FUNCTION_BLOCK oven (* ODE *)
  (* Standard: 61499-2 *)
  (* Version 0.1, 2017-00-25, hpea485, UOA *)
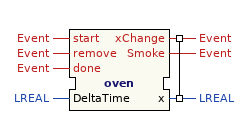
  EVENT_INPUT
    start;
    remove;
    done;
  END_EVENT
  EVENT_OUTPUT
    xChange WITH x;
    Smoke;
  END_EVENT
  VAR_INPUT
    DeltaTime : LREAL := 0.01;
  END_VAR
  VAR_OUTPUT
    x : LREAL;
  END_VAR
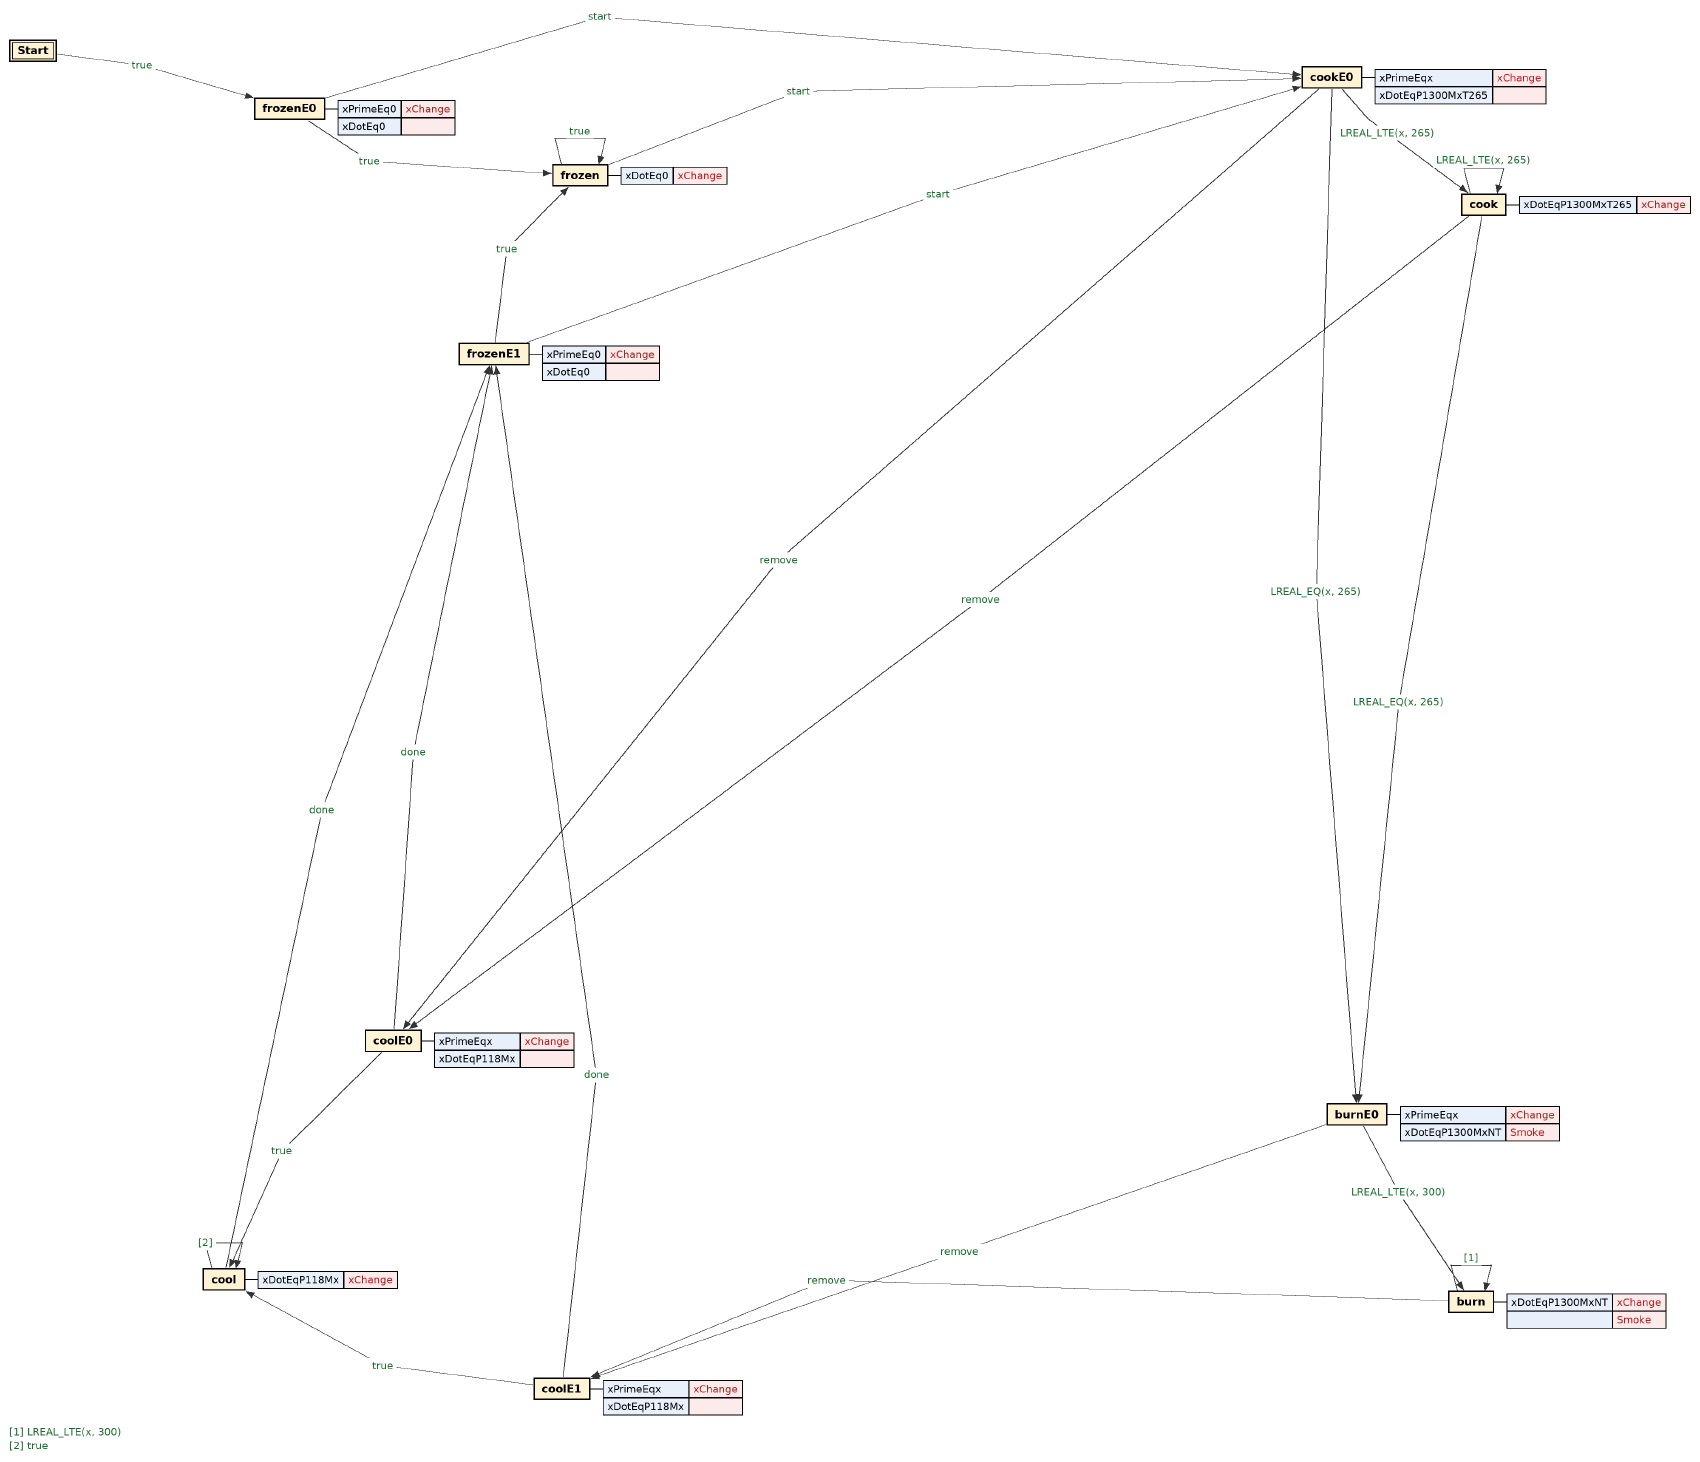
  EC_STATES
    Start;
    frozenE0 : xPrimeEq0 -> xChange, xDotEq0;
    frozen : xDotEq0 -> xChange;
    cookE0 : xPrimeEqx -> xChange, xDotEqP1300MxT265;
    cook : xDotEqP1300MxT265 -> xChange;
    burnE0 : xPrimeEqx -> xChange, xDotEqP1300MxNT -> Smoke;
    burn : xDotEqP1300MxNT -> xChange, -> Smoke;
    coolE0 : xPrimeEqx -> xChange, xDotEqP118Mx;
    coolE1 : xPrimeEqx -> xChange, xDotEqP118Mx;
    cool : xDotEqP118Mx -> xChange;
    frozenE1 : xPrimeEq0 -> xChange, xDotEq0;
  END_STATES
  EC_TRANSITIONS
    Start TO frozenE0 := true;
    frozenE0 TO cookE0 := start;
    frozenE0 TO frozen := true;
    frozen TO cookE0 := start;
    frozen TO frozen := true;
    cookE0 TO coolE0 := remove;
    cookE0 TO burnE0 := LREAL_EQ(x, 265);
    cookE0 TO cook := LREAL_LTE(x, 265);
    cook TO coolE0 := remove;
    cook TO burnE0 := LREAL_EQ(x, 265);
    cook TO cook := LREAL_LTE(x, 265);
    burnE0 TO coolE1 := remove;
    burnE0 TO burn := LREAL_LTE(x, 300);
    burn TO coolE1 := remove;
    burn TO burn := LREAL_LTE(x, 300);
    coolE0 TO frozenE1 := done;
    coolE0 TO cool := true;
    coolE1 TO frozenE1 := done;
    coolE1 TO cool := true;
    cool TO frozenE1 := done;
    cool TO cool := true;
    frozenE1 TO cookE0 := start;
    frozenE1 TO frozen := true;
  END_TRANSITIONS
  ALGORITHM xPrimeEq0 IN C: (* ODE_init *)
x_prime = 0;
  END_ALGORITHM
  ALGORITHM xPrimeEqx IN C: (* ODE_init *)
x_prime = x;
  END_ALGORITHM
  ALGORITHM xDotEq0 IN C: (* ODE *)
x_dot = 0;
  END_ALGORITHM
  ALGORITHM xDotEqP1300MxT265 IN C: (* ODE *)
x_dot = 0.1 * (300 - x);
x_trigger = 265;
  END_ALGORITHM
  ALGORITHM xDotEqP118Mx IN C: (* ODE *)
x_dot = 0.1 * (18 - x);
  END_ALGORITHM
  ALGORITHM xDotEqP1300MxNT IN C: (* ODE *)
x_dot = 0.1 * (300 - x);
  END_ALGORITHM
END_FUNCTION_BLOCK
